(*			
	RafalOS
	Rafał Osajda		20.11.2025		TC 4024.66
	Moduł przygotowania danych dla Okna diagramu we wszystkich trybach
*)
FUNCTION_BLOCK FB_MCHMIPrepareDataForScreen_06_XX EXTENDS FB_MCHMIPrepareDataForScreen IMPLEMENTS ITF_MCHMIPrepareDataForScreen
VAR
	itfMachineControlHMI	: ITF_MCHMIMachineControl_HMI_PrepScr_06_XX;
	refstData				: REFERENCE TO ST_MCHMIPrepareScreen_06_XX;
END_VAR

(*			
	RafalOS
	Rafał Osajda		19.11.2025		TC 4024.66
	Czyści danych przy zmienia ramki po poprzedniej ramce
*)
METHOD PUBLIC ClearAfterScreen : BOOL
VAR_INPUT
END_VAR
SUPER^.ClearAfterScreen ();
END_METHOD

METHOD PUBLIC LinkDataHMI_06_XX : BOOL
VAR_INPUT
	refstData				: REFERENCE TO ST_MCHMIPrepareScreen_06_XX;
END_VAR
THIS^.refstData REF= refstData;
END_METHOD

METHOD PUBLIC LinkMachineControlHMI : BOOL
VAR_INPUT
	fbMachineControlHMI	: ITF_MCHMIMachineControl_HMI_PrepScr_06_XX;
END_VAR
this^.itfMachineControlHMI := fbMachineControlHMI;
END_METHOD

(*			
	RafalOS
	Rafał Osajda		14.11.2025		TC 4024.66
	Metoda przygotowywania danych dla HMI 
	W niej odbywa się odpytywanie właściego elementu przez łącznik
*)
METHOD PUBLIC PrepareDataForHMI : BOOL
VAR_INPUT
END_VAR
SUPER^.PrepareDataForHMI ();
END_METHOD

(*			
	RafalOS
	Rafał Osajda		19.11.2025		TC 4024.66
	Przygotowanie ramki pood tamke do wyświetlenia - tylko przygotowanie a nie przygotowanie danych do wyświetlenia
*)
METHOD PUBLIC PrepareForScreen : BOOL
VAR_INPUT
END_VAR
SUPER^.PrepareForScreen ();
END_METHOD

END_FUNCTION_BLOCK

(* stored: Version 1.1.0.1
   POU FB_MCHMIPrepareDataForScreen_06_XX: Id {d9ab5ce6-fe70-0537-3653-306a1d96a255}, SpecialFunc None
   Folder ITF_PDFS: Id {77bdb900-4748-0c69-1777-5a93fb82f601}
   Method ClearAfterScreen: Id {7e29f3c8-32dc-0e9b-0dd5-360a6a118200}
   Method LinkDataHMI_06_XX: Id {7ba8154e-6f52-018b-1a4b-e41c8b40008e}
   Method LinkMachineControlHMI: Id {9ff87962-8c61-02a3-2181-3d9f6e3a6623}
   Method PrepareDataForHMI: Id {2595d879-11d4-08a2-31e5-37340d685f33}
   Method PrepareForScreen: Id {c586df67-c716-0c6a-238f-1f6286330427} *)
